# B&R Automation Studio project Steppermotor_withx20
Automation Studio 4.7.3.93 SP; technology packages: mappMotion 5.10.1, mappSafety 5.10.1

## Configuration Config1

CPU X20CP1382, AutomationRuntime C4.72, Build 4.1.2, Safety 0.0, Vc V4.72.0

### Task classes (Cpu.sw)
```
Cyclic#1 (cycle 2000 us, tolerance 0 us):
  Program <- Program.prg
Libraries: McBase, MpAxis, McAxis, MpBase, McAcpAx, McStpAx
```

### Hardware
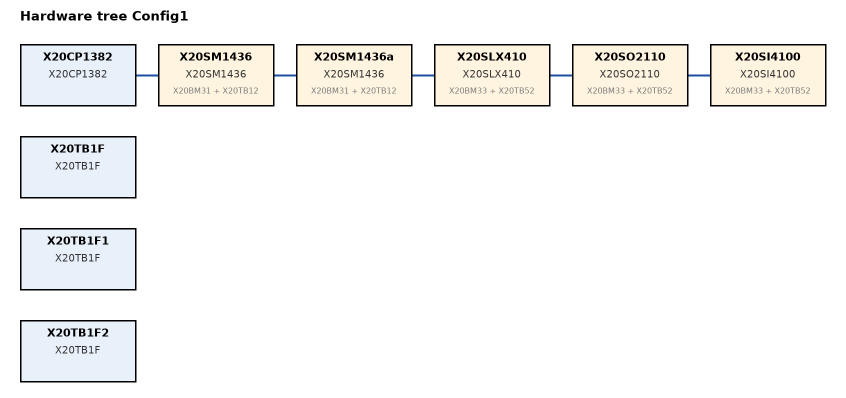
```
X20BM31 : X20BM31 v1.0.0.1  [X2X1 -> X20CP1382.IF6]
X20BM31a : X20BM31 v1.0.0.1  [X2X1 -> X20BM31.X2X2]
X20BM33 : X20BM33 v1.0.0.6  [X2X1 -> X20BM31a.X2X2]
X20BM33a : X20BM33 v1.0.0.6  [X2X1 -> X20BM33.X2X2]
X20BM33b : X20BM33 v1.0.0.6  [X2X1 -> X20BM33a.X2X2]
X20CP1382 : X20CP1382 v1.11.0.0  [X1 -> X1.SL; X2 -> X2.SL; X3 -> X3.SL]
  Module X1 (Type=X1, Virtual=true, Version=1.11.0.0)
    Connection (Connector=SS1, TargetModule=X20TB1F, TargetConnector=SS)
    Connection (Connector=SL, TargetModule=X20CP1382, TargetConnector=X1)
  Module X2 (Type=X2, Virtual=true, Version=1.11.0.0)
    Connection (Connector=SS1, TargetModule=X20TB1F1, TargetConnector=SS)
    Connection (Connector=SL, TargetModule=X20CP1382, TargetConnector=X2)
  Module X3 (Type=X3, Virtual=true, Version=1.11.0.0)
    Connection (Connector=SS1, TargetModule=X20TB1F2, TargetConnector=SS)
    Connection (Connector=SL, TargetModule=X20CP1382, TargetConnector=X3)
  Connector IF2:
    ActivateDevice = 1
    Mode = Manual
    InternetAddress = 192.168.1.10
    SubnetMask = 255.255.255.0
  ConfigurationID = Steppermotor_withx20_Config1
  TimerDeviceType = EPLX2X
  TimerDevice = X20CP1382.IF6
  Cyclic1Duration = 2000
  Cyclic1Tolerance = 0
X20SI4100 : X20SI4100 v2.2.0.1  [SS1 -> X20TB52b.SS; SL -> X20BM33b.SL1]
  SafeModuleID = 3
X20SLX410 : X20SLX410 v2.2.0.0  [SS1 -> X20TB52.SS; SL -> X20BM33.SL1]
X20SM1436 : X20SM1436 v2.2.0.0  [SS1 -> X20TB12.SS; SL -> X20BM31.SL1]
  FunctionModel/DriveConfiguration:
    ModuleParameters = StepperParameters
  FunctionModel/DriveConfiguration/ModuleParameters:
    McStepperTypeID = X20Config
    EncoderType = Incremental
    ReferencePulse = yes
    RatedCurrent = 3.0
    MaximumCurrent = 3.51
    AxesNumber = 1
    FullStepThreshold = 1
    StallDetection = 1
    SmartCurrentControl = 0
    BrakeOutput = 0
    NumberOfDigitalInputs = 3
    NumberOfTriggers = 1
  FunctionModel/DriveConfiguration/Channel[1]/RealAxis:
    AxisReference = gAxis_1
  FunctionModel/DriveConfiguration/Channel[1]/RealAxis/MechanicalElements/Gearbox:
    InputIsReadOnly = 0
    Input = 1
    OutputIsReadOnly = 0
    Output = 1
  FunctionModel/DriveConfiguration/Channel[1]/RealAxis/MechanicalElements/RotaryToLinearTransformation:
    ReferenceDistanceIsReadOnly = 0
    ReferenceDistance = 1
  FunctionModel/DriveConfiguration/Channel[1]/RealAxis/Motor:
    SteppingAngle = 1.8
  FunctionModel/DriveConfiguration/Channel[1]/RealAxis:
    EncoderLink = NoEncoder
  FunctionModel/DriveConfiguration/Channel[1]/RealAxis/Controller:
    ModeIsReadOnly = 0
    Mode = PositionAndCurrentController
  FunctionModel/DriveConfiguration/Channel[1]/RealAxis/Controller/Mode/Current:
    StandstillCurrent = 0.09
    ConstantSpeedCurrent = 0.45
    SpeedChangeCurrent = 0.9
    FullStepThreshold = 0.0
    MotorSettlingTime = 1
    DelayedCurrentSwitchOff = 1
  FunctionModel/DriveConfiguration/Channel[1]/RealAxis/Controller/Mode/Position:
    ProportionalGain = 20.0
    MaximumProportionalAction = 1e10
    PredictionTime = 0.01
    TotalDelayTime = 0.01
  FunctionModel/DriveConfiguration/Channel[1]/RealAxis/Homing:
    Mode = Direct
  FunctionModel/DriveConfiguration/Channel[1]/RealAxis/Homing/Mode:
    Position = 0.0
    ReferencePulse = NotUsed
  FunctionModel/DriveConfiguration/Channel[1]/RealAxis/Homing:
    RestorePositionVariable = 
  FunctionModel/DriveConfiguration/Channel[1]/RealAxis/StopReaction:
    DriveError = DecelerationLimit
  FunctionModel/DriveConfiguration/Channel[1]/RealAxis/MovementErrorLimits:
    PositionError = 1.0
    StallDetectionConfiguration = NotUsed
  FunctionModel/DriveConfiguration/Channel[1]/RealAxis:
    JerkFilter = NotUsed
  FunctionModel/DriveConfiguration/Channel[1]/RealAxis/DigitalInputs/HomingSwitch:
    Source = NotUsed
    Level = High
  FunctionModel/DriveConfiguration/Channel[1]/RealAxis/DigitalInputs/PositiveLimitSwitch:
    Source = NotUsed
    Level = High
  FunctionModel/DriveConfiguration/Channel[1]/RealAxis/DigitalInputs/NegativeLimitSwitch:
    Source = NotUsed
    Level = High
  FunctionModel/DriveConfiguration/Channel[1]/RealAxis/DigitalInputs/Trigger1:
    Source = NotUsed
    Level = High
  FunctionModel/DriveConfiguration/Channel[1]/RealAxis/DigitalInputs/Trigger2:
    Source = NotUsed
    Level = High
  FunctionModel/DriveConfiguration/Channel[1]/RealAxis/DigitalInputs/Quickstop:
    Input = NotUsed
  FunctionModel/DriveConfiguration/Channel[1]/RealAxis/DigitalOutputs:
    BrakeControl = NotUsed
X20SM1436a : X20SM1436 v2.2.0.0  [SS1 -> X20TB12a.SS; SL -> X20BM31a.SL1]
  FunctionModel/DriveConfiguration:
    ModuleParameters = StepperParameters
  FunctionModel/DriveConfiguration/ModuleParameters:
    McStepperTypeID = X20Config
    EncoderType = Incremental
    ReferencePulse = yes
    RatedCurrent = 3.0
    MaximumCurrent = 3.51
    AxesNumber = 1
    FullStepThreshold = 1
    StallDetection = 1
    SmartCurrentControl = 0
    BrakeOutput = 0
    NumberOfDigitalInputs = 3
    NumberOfTriggers = 1
  FunctionModel/DriveConfiguration/Channel[1]/RealAxis:
    AxisReference = 
  FunctionModel/DriveConfiguration/Channel[1]/RealAxis/MechanicalElements/Gearbox:
    InputIsReadOnly = 0
    Input = 1
    OutputIsReadOnly = 0
    Output = 1
  FunctionModel/DriveConfiguration/Channel[1]/RealAxis/MechanicalElements/RotaryToLinearTransformation:
    ReferenceDistanceIsReadOnly = 0
    ReferenceDistance = 1
  FunctionModel/DriveConfiguration/Channel[1]/RealAxis/Motor:
    SteppingAngle = 1.8
  FunctionModel/DriveConfiguration/Channel[1]/RealAxis:
    EncoderLink = NoEncoder
  FunctionModel/DriveConfiguration/Channel[1]/RealAxis/Controller:
    ModeIsReadOnly = 0
    Mode = CurrentController
  FunctionModel/DriveConfiguration/Channel[1]/RealAxis/Controller/Mode/Current:
    StandstillCurrent = 0.09
    ConstantSpeedCurrent = 0.45
    SpeedChangeCurrent = 0.9
    FullStepThreshold = 0.0
    MotorSettlingTime = 1
    DelayedCurrentSwitchOff = 1
  FunctionModel/DriveConfiguration/Channel[1]/RealAxis/Homing:
    Mode = Direct
  FunctionModel/DriveConfiguration/Channel[1]/RealAxis/Homing/Mode:
    Position = 0.0
    ReferencePulse = NotUsed
  FunctionModel/DriveConfiguration/Channel[1]/RealAxis/Homing:
    RestorePositionVariable = 
  FunctionModel/DriveConfiguration/Channel[1]/RealAxis/StopReaction:
    DriveError = DecelerationLimit
  FunctionModel/DriveConfiguration/Channel[1]/RealAxis/MovementErrorLimits:
    PositionError = 1.0
    StallDetectionConfiguration = NotUsed
  FunctionModel/DriveConfiguration/Channel[1]/RealAxis:
    JerkFilter = NotUsed
  FunctionModel/DriveConfiguration/Channel[1]/RealAxis/DigitalInputs/HomingSwitch:
    Source = NotUsed
    Level = High
  FunctionModel/DriveConfiguration/Channel[1]/RealAxis/DigitalInputs/PositiveLimitSwitch:
    Source = NotUsed
    Level = High
  FunctionModel/DriveConfiguration/Channel[1]/RealAxis/DigitalInputs/NegativeLimitSwitch:
    Source = NotUsed
    Level = High
  FunctionModel/DriveConfiguration/Channel[1]/RealAxis/DigitalInputs/Trigger1:
    Source = NotUsed
    Level = High
  FunctionModel/DriveConfiguration/Channel[1]/RealAxis/DigitalInputs/Trigger2:
    Source = NotUsed
    Level = High
  FunctionModel/DriveConfiguration/Channel[1]/RealAxis/DigitalInputs/Quickstop:
    Input = NotUsed
  FunctionModel/DriveConfiguration/Channel[1]/RealAxis/DigitalOutputs:
    BrakeControl = NotUsed
X20SO2110 : X20SO2110 v2.2.0.1  [SS1 -> X20TB52a.SS; SL -> X20BM33a.SL1]
X20TB12 : X20TB12 v1.0.0.0
X20TB12a : X20TB12 v1.0.0.0
X20TB1F : X20TB1F v1.0.0.0
X20TB1F1 : X20TB1F v1.0.0.0
X20TB1F2 : X20TB1F v1.0.0.0
X20TB52 : X20TB52 v1.0.0.1
X20TB52a : X20TB52 v1.0.0.1
X20TB52b : X20TB52 v1.0.0.1
```

### Config_1.axis - X20CP1382/mappMotion/Config_1.axis
```
Element gAxis_1 (Type=axis)
  BaseTypeIsReadOnly = 0
  BaseType = Rotary
    MeasurementUnitIsReadOnly = 0
    MeasurementUnit = 17476
    MeasurementResolutionIsReadOnly = 0
    MeasurementResolution = 0.01
    CountDirectionIsReadOnly = 0
    CountDirection = Standard
  MovementLimitsIsReadOnly = 0
  MovementLimits = Internal
    Position:
      LowerLimitMin = -1.79769313486231E308
      UpperLimitMax = 1.79769313486231E308
      LowerLimit = -1000.0
      UpperLimit = 1000.0
    VelocityIsReadOnly = 0
    Velocity:
      VelocityMax = 3.4E38
      Velocity = 10.0
    AccelerationIsReadOnly = 0
    Acceleration:
      AccelerationMax = 3.4E38
      Acceleration = 50.0
    DecelerationIsReadOnly = 0
    Deceleration:
      DecelerationMax = 3.4E38
      Deceleration = 50.0
  Alarms = None
```

- Safety project (password-protected, skipped)

## Logical view

Binary libraries used (declarations not repeated): operator, runtime, astime, AsIecCon, McBase 5.10.1, MpAxis 5.10.1, McAxis 5.10.1, MpBase, McAcpAx 5.10.1, McStpAx


### Program Logical/Program (IEC)

#### Variables.var
```iecst
VAR
	MpAxisBasic_0 : MpAxisBasic;
	AxisParameters : MpAxisBasicParType;
END_VAR
```

#### Main.st
```iecst
PROGRAM _INIT

	MpAxisBasic_0.MpLink := ADR(gAxis_1);
	MpAxisBasic_0.Enable := TRUE;
	MpAxisBasic_0.Parameters := ADR(AxisParameters);

	AxisParameters.Position := 100.0;
	AxisParameters.Velocity := 10.0;
	AxisParameters.Acceleration := 50.0;
	AxisParameters.Deceleration := 50.0;

END_PROGRAM

PROGRAM _CYCLIC

	//MpAxisBasic_0();

END_PROGRAM

PROGRAM _EXIT

	MpAxisBasic_0.Power  := FALSE;
	MpAxisBasic_0.Home   := FALSE;
	MpAxisBasic_0.MoveAbsolute := FALSE;
	MpAxisBasic_0.MoveAdditive := FALSE;
	MpAxisBasic_0.MoveVelocity := FALSE;
	MpAxisBasic_0.Stop         := FALSE;
	MpAxisBasic_0.ErrorReset   := FALSE;
	MpAxisBasic_0();

	MpAxisBasic_0.Enable := FALSE;
	MpAxisBasic_0();

END_PROGRAM
```

Listed in the project but not available here: Logical/Global.typ, Logical/Global.var
